// TIA Portal project "PLC" (V15.1)

(* hardware
DEVICE "S7-1200 station_1"  S7-1200 Station
   slot 0: "Rack_0"  S7-1200 Rack  Rack  V1.0
   slot 1: "PLC_1"  CPU 1214C DC/DC/DC  6ES7 214-1AG40-0XB0  V4.2
DEVICE "HMI_1"  KTP700 Basic PN
   slot 0: "HMI_1"  KTP700 Basic PN  6AV2 123-2GB03-0AX0  15.1.0.0
   slot 1: "HMI_RT_1"  KTP700 Basic PN  6AV2 123-2GB03-0AX0  15.1.0.0
   slot 5: "HMI_1.IE_CP_1"  PROFINET Interface  15.0.1.0
      slot 1: "PROFINET Interface_1"  PROFINET Interface
         slot 1: "Port_1"  Port
*)

// ===== PLC "PLC_1"  CPU 1214C DC/DC/DC =====

VAR_GLOBAL   // PLC tag table "默认变量表"
   "物料到位信号" AT %I0.0 : Bool;
   "物料检测信号" AT %I0.6 : Bool;
   "传送带正转信号" AT %Q0.1 : Bool;
   "推料动作" AT %Q0.4 : Bool;
   "运行步骤" AT %MW100 : Int;
   "物资发放" AT %M22.7 : Bool;
END_VAR

DATA_BLOCK "人脸语音通讯"   // DB9
{ S7_Optimized_Access := 'TRUE' }
VERSION : 0.1
   VAR
      re_data : Array[0..31] of Byte;
      use_data : Array[0..31] of String;
      empty_data : Array[0..31] of Byte;
      人脸语音通讯成功 : Bool;
   END_VAR
BEGIN
END_DATA_BLOCK

DATA_BLOCK "图像识别通讯"   // DB12
{ S7_Optimized_Access := 'TRUE' }
VERSION : 0.1
   VAR
      re_data : Array[0..31] of Byte;
      use_data : Array[0..31] of String;
      empty_data : Array[0..31] of Byte;
      tx_data : Array[0..31] of Byte;
      人员1信息 : Array[0..6] of String;
      人员2信息 : Array[0..6] of String;
      人员3信息 : Array[0..6] of String;
      人员4信息 : Array[0..6] of String;
      人员5信息 : Array[0..6] of String;
      人员6信息 : Array[0..6] of String;
      图像识别发送标志位 : Bool;
      图像识别通讯成功 : Bool;
   END_VAR
BEGIN
END_DATA_BLOCK

DATA_BLOCK "视觉通讯"   // DB15
{ S7_Optimized_Access := 'TRUE' }
VERSION : 0.1
   VAR
      re_data : Array[0..310] of Byte;
      use_data : Array[0..100] of String;
      empty_data : Array[0..310] of Byte;
      tx_data : Array[0..310] of Byte;
      发送数据的长度 : Int;
      视觉发送标志位 : Bool;
      视觉通讯成功 : Bool;
      A地区状态 : String;
      B地区状态 : String;
      C地区状态 : String;
      D地区状态 : String;
   END_VAR
BEGIN
END_DATA_BLOCK

DATA_BLOCK "机器人通讯"   // DB18
{ S7_Optimized_Access := 'TRUE' }
VERSION : 0.1
   VAR
      re_data : Array[0..31] of Byte;
      use_data : Array[0..31] of String;
      empty_data : Array[0..31] of Byte;
      tx_data : Array[0..31] of Byte;
      机器人发送标志位 : Bool;
      机器人通讯成功 : Bool;
      二维码分类计数 : Int;
   END_VAR
BEGIN
END_DATA_BLOCK

// folder: System blocks/Program resources

DATA_BLOCK "PLC_1_Receive_DB"   // DB1
{ S7_Optimized_Access := 'TRUE' }
AUTHOR : SIMATIC
FAMILY : MC7Plus
NAME : TC_IP_v4
VERSION : 1.0
// stored: InstanceOfName TCON_IP_v4
"TCON_IP_v4"
BEGIN
   ID := 1;
   InterfaceId := 64;
   LocalPort := 4001;
END_DATA_BLOCK

DATA_BLOCK "PLC_1_Receive_DB_1"   // DB2
{ S7_Optimized_Access := 'TRUE' }
AUTHOR : SIMATIC
FAMILY : MC7Plus
NAME : TC_IP_v4
VERSION : 1.0
// stored: InstanceOfName TCON_IP_v4
"TCON_IP_v4"
BEGIN
   ID := 2;
   InterfaceId := 64;
   LocalPort := 2005;
END_DATA_BLOCK

DATA_BLOCK "PLC_1_Receive_DB_2"   // DB3
{ S7_Optimized_Access := 'TRUE' }
AUTHOR : SIMATIC
FAMILY : MC7Plus
NAME : TC_IP_v4
VERSION : 1.0
// stored: InstanceOfName TCON_IP_v4
"TCON_IP_v4"
BEGIN
   ID := 3;
   InterfaceId := 64;
   LocalPort := 3001;
END_DATA_BLOCK

DATA_BLOCK "PLC_1_Receive_DB_3"   // DB4
{ S7_Optimized_Access := 'TRUE' }
AUTHOR : SIMATIC
FAMILY : MC7Plus
NAME : TC_IP_v4
VERSION : 1.0
// stored: InstanceOfName TCON_IP_v4
"TCON_IP_v4"
BEGIN
   ID := 4;
   InterfaceId := 64;
   LocalPort := 2001;
END_DATA_BLOCK

DATA_BLOCK "延时函数"   // DB13
{ S7_Optimized_Access := 'TRUE' }
AUTHOR : Simatic
FAMILY : IEC
NAME : IEC_TMR
VERSION : 1.0
// stored: InstanceOfName IEC_TIMER
"IEC_TIMER"
BEGIN
END_DATA_BLOCK

// folder: (top level)

FUNCTION "发送" : Void   // FC2, SCL
{ S7_Optimized_Access := 'TRUE' }
VERSION : 0.1
   VAR_INPUT
      buf : String;
      num : Int;
   END_VAR
   VAR_TEMP
      strlen : Int;
   END_VAR
BEGIN
   //字符串转换成字符指令
   "视觉通讯".发送数据的长度 := LEN(#buf);
   IF #num = 2 THEN
       Strg_TO_Chars(Strg := #buf,  //需要转换的字符串
                     pChars := 0,    //字符数组的起始位置
                     Cnt => #strlen, // 转成成功的长度，储存到
                     Chars := "图像识别通讯".tx_data);//字符串的数组
       "图像识别通讯".图像识别发送标志位 := 1;
   ELSIF #num = 3 THEN
       Strg_TO_Chars(Strg := #buf,
                     pChars := 0,
                     Cnt => #strlen,
                     Chars := "视觉通讯".tx_data);
       "视觉通讯".视觉发送标志位 := 1;
   ELSIF #num = 4 THEN
       Strg_TO_Chars(Strg := #buf,
                     pChars := 0,
                     Cnt => #strlen,
                     Chars := "机器人通讯".tx_data);
       "机器人通讯".机器人发送标志位 := 1;
   END_IF;
END_FUNCTION

FUNCTION "图像识别通讯主程序" : Void   // FC4, LAD
{ S7_Optimized_Access := 'TRUE' }
VERSION : 0.1
   VAR_TEMP
      i : Int;
      i_1 : Int;
      i_2 : Int;
      send_data : String;
   END_VAR
BEGIN

REGION Network 1
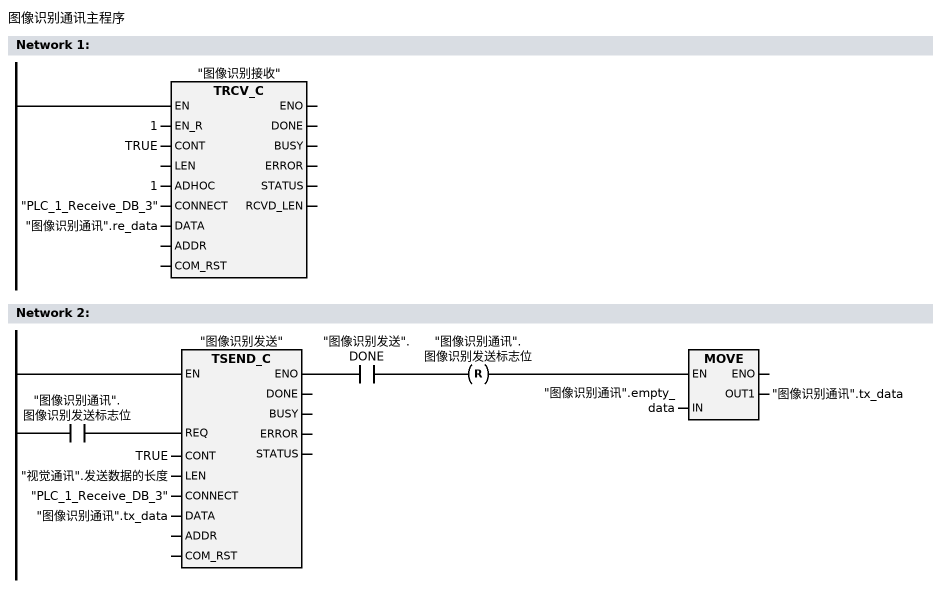
   "图像识别接收"(EN_R := 1, CONT := TRUE, ADHOC := 1, CONNECT := "PLC_1_Receive_DB_3", DATA := "图像识别通讯".re_data);   // TRCV_C
END_REGION

REGION Network 2
   // ENO of a box is taken as its EN; it also drops when the box reports an error
   "图像识别发送"(REQ := "图像识别通讯".图像识别发送标志位,   // TSEND_C
            CONT := TRUE,
            LEN := "视觉通讯".发送数据的长度,
            CONNECT := "PLC_1_Receive_DB_3",
            DATA := "图像识别通讯".tx_data);
   IF "图像识别发送".DONE THEN
       "图像识别通讯".图像识别发送标志位 := FALSE;
       "图像识别通讯".tx_data := "图像识别通讯".empty_data;
   END_IF;
END_REGION

REGION Network 3 (SCL)
   IF "图像识别接收".DONE THEN
       //字符分割函数
       FOR #i := 0 TO 31 DO
           IF "图像识别通讯".re_data[#i] = ',' OR "图像识别通讯".re_data[#i] = 16#0 THEN
               Chars_TO_Strg(Chars := "图像识别通讯".re_data,
                             pChars := #i_1,
                             Cnt := #i - #i_1,
                             Strg => "图像识别通讯".use_data[#i_2]);
               #i_1 := #i + 1;
               #i_2 += 1;
           END_IF;
       END_FOR;
       "图像识别通讯".re_data := "图像识别通讯".empty_data;

       FOR #i := 0 TO 2 DO
           IF "图像识别通讯".use_data[0] = "图像识别通讯"."人员1信息"[#i + 2] THEN
               "发送"(buf := 'D1',
                    num := 4);
               EXIT;
           END_IF;
           IF "图像识别通讯".use_data[0] = "图像识别通讯"."人员2信息"[#i + 2] THEN
               //"视觉通讯"."2号人员信息"[#i + 2] := ' ';
               "发送"(buf := 'A1',
                     num := 4);
               EXIT;
           END_IF;
           IF "图像识别通讯".use_data[0] = "图像识别通讯"."人员3信息"[#i + 2] THEN
               //"视觉通讯"."3号人员信息"[#i + 2] := ' ';
               "发送"(buf := 'B1',
                    num := 4);
               EXIT;
           END_IF;
           IF "图像识别通讯".use_data[0] = "图像识别通讯"."人员4信息"[#i + 2] THEN
               //"视觉通讯"."4号人员信息"[#i + 2] := ' ';
               "发送"(buf := 'C1',
                    num := 4);
               EXIT;
           END_IF;
       END_FOR;
   END_IF;
END_REGION
END_FUNCTION

FUNCTION "机器人通讯主程序" : Void   // FC5, LAD
{ S7_Optimized_Access := 'TRUE' }
VERSION : 0.1
   VAR_TEMP
      i : Int;
      i_1 : Int;
      i_2 : Int;
      ab : String;
   END_VAR
BEGIN

REGION Network 1
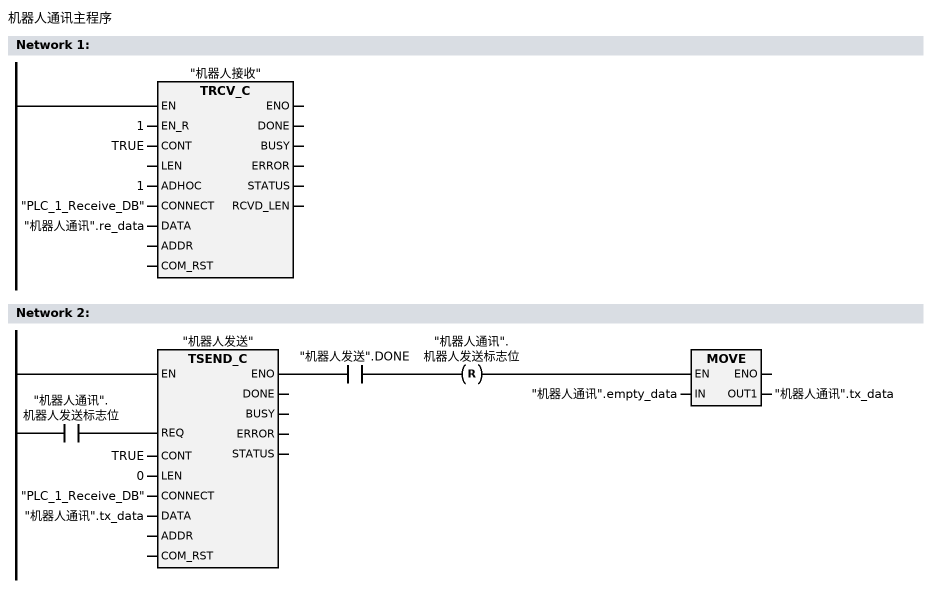
   "机器人接收"(EN_R := 1, CONT := TRUE, ADHOC := 1, CONNECT := "PLC_1_Receive_DB", DATA := "机器人通讯".re_data);   // TRCV_C
END_REGION

REGION Network 2
   // ENO of a box is taken as its EN; it also drops when the box reports an error
   "机器人发送"(REQ := "机器人通讯".机器人发送标志位,   // TSEND_C
           CONT := TRUE,
           LEN := 0,
           CONNECT := "PLC_1_Receive_DB",
           DATA := "机器人通讯".tx_data);
   IF "机器人发送".DONE THEN
       "机器人通讯".机器人发送标志位 := FALSE;
       "机器人通讯".tx_data := "机器人通讯".empty_data;
   END_IF;
END_REGION

REGION Network 3 (SCL)
   IF "机器人接收".DONE THEN
       //字符分割函数
       FOR #i := 0 TO 31 DO
           IF "机器人通讯".re_data[#i] = ',' OR "机器人通讯".re_data[#i] = 16#0 THEN
               Chars_TO_Strg(Chars := "机器人通讯".re_data,
                             pChars := #i_1,
                             Cnt := #i - #i_1,
                             Strg => "机器人通讯".use_data[#i_2]);
               #i_1 := #i + 1;
               #i_2 += 1;
           END_IF;
       END_FOR;
       "机器人通讯".re_data := "机器人通讯".empty_data;
       //二维码分类
       IF "机器人通讯".use_data[0] = 'ok1' THEN
           "发送"(buf := 'ewm',
                num := 3);
       ELSIF "机器人通讯".use_data[0] = 'ok2' THEN
           IF "机器人通讯".二维码分类计数 > 4 THEN
               ;
           ELSE
               "机器人通讯".二维码分类计数 += 1;
               "发送"(buf := 'set',
                    num := 4);
           END_IF;
       ELSIF "机器人通讯".use_data[0] = 'run' THEN
           "物资发放" := 1;
       END_IF;
   END_IF;
END_REGION
END_FUNCTION

FUNCTION "视觉通讯主程序" : Void   // FC6, LAD
{ S7_Optimized_Access := 'TRUE' }
VERSION : 0.1
   VAR_TEMP
      i : Int;
      i_1 : Int;
      i_2 : Int;
   END_VAR
BEGIN

REGION Network 1
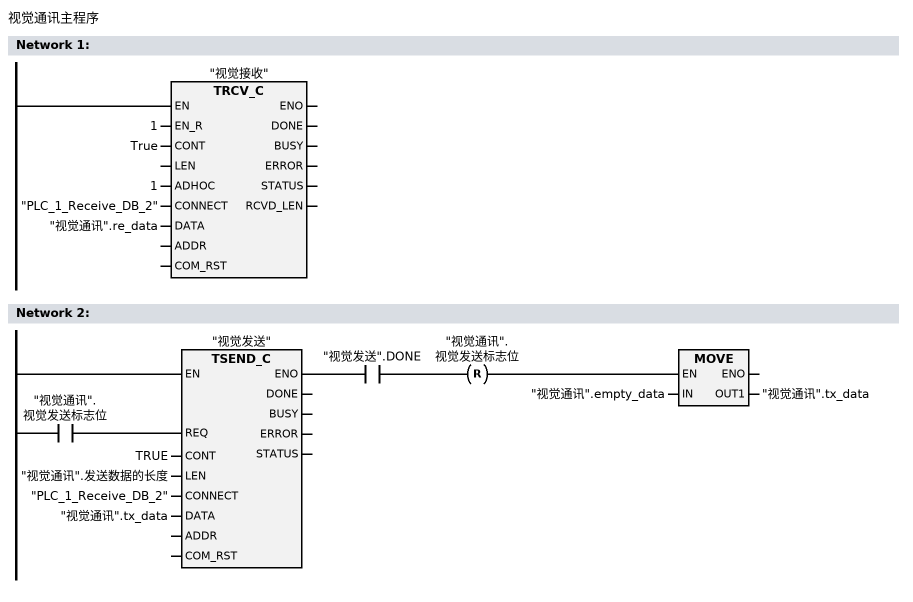
   "视觉接收"(EN_R := 1, CONT := True, ADHOC := 1, CONNECT := "PLC_1_Receive_DB_2", DATA := "视觉通讯".re_data);   // TRCV_C
END_REGION

REGION Network 2
   // ENO of a box is taken as its EN; it also drops when the box reports an error
   "视觉发送"(REQ := "视觉通讯".视觉发送标志位,   // TSEND_C
          CONT := TRUE,
          LEN := "视觉通讯".发送数据的长度,
          CONNECT := "PLC_1_Receive_DB_2",
          DATA := "视觉通讯".tx_data);
   IF "视觉发送".DONE THEN
       "视觉通讯".视觉发送标志位 := FALSE;
       "视觉通讯".tx_data := "视觉通讯".empty_data;
   END_IF;
END_REGION

REGION Network 3 (SCL)
   IF "视觉接收".DONE THEN
       //字符分割函数
       FOR #i := 0 TO 310 DO
           IF "视觉通讯".re_data[#i] = ',' OR "视觉通讯".re_data[#i] = 16#0 THEN
               Chars_TO_Strg(Chars := "视觉通讯".re_data,
                             pChars := #i_1,
                             Cnt := #i - #i_1,
                             Strg => "视觉通讯".use_data[#i_2]);
               #i_1 := #i + 1;
               #i_2 += 1;
           END_IF;
       END_FOR;
       "视觉通讯".re_data := "视觉通讯".empty_data;

       //处理地图信息

       IF "视觉通讯".use_data[0] = '{name:Tom;active:A;drink:kuangquanshui;food:fangbianmian;supplies:xifashui}' THEN
           "图像识别通讯".人员1信息[0] := 'Tom';
           "图像识别通讯".人员1信息[1] := 'A';
           "图像识别通讯".人员1信息[2] := 'kuangquanshui';
           "图像识别通讯".人员1信息[3] := 'fangbianmian';
           "图像识别通讯".人员1信息[4] := 'xifashui';
           "发送"(buf := 'D1',
                num := 4);
       ELSIF "视觉通讯".use_data[0] = '{name:Jack;active:B;drink:kele;food:pingguo;supplies:maojin}' THEN
           "图像识别通讯".人员2信息[0] := 'Jack';
           "图像识别通讯".人员2信息[1] := 'B';
           "图像识别通讯".人员2信息[2] := 'kele';
           "图像识别通讯".人员2信息[3] := 'pingguo';
           "图像识别通讯".人员2信息[4] := 'maojin';
           "发送"(buf:='A1',
                num:= 4);

           //处理物资的坐标信息

       ELSIF "视觉通讯".use_data[0] = '{name:Andy;active:C;drink:fenda;food:mianbao;supplies:yagao}' THEN
           "图像识别通讯".人员3信息[0] := 'Andy';
           "图像识别通讯".人员3信息[1] := 'C';
           "图像识别通讯".人员3信息[2] := 'fenda';
           "图像识别通讯".人员3信息[3] := 'mianbao';
           "图像识别通讯".人员3信息[4] := 'yagao';
           "发送"(buf := 'B1',
                num := 4);
       ELSIF "视觉通讯".use_data[0] = '{name:Vicky;active:D;drink:xuebi;food:guantou;supplies:zhijin}' THEN
           "图像识别通讯".人员4信息[0] := 'Vicky';
           "图像识别通讯".人员4信息[1] := 'D';
           "图像识别通讯".人员4信息[2] := 'xuebi';
           "图像识别通讯".人员4信息[3] := 'guantou';
           "图像识别通讯".人员4信息[4] := 'zhijin';
           "发送"(buf := 'C1',
                num := 4);
       ELSIF "视觉通讯".use_data[0] = '{name:Cindy;active:E;drink:hongniu;food:mangguo;supplies:tuoxie}' THEN
           "图像识别通讯".人员5信息[0] := 'Cindy';
           "图像识别通讯".人员5信息[1] := 'E';
           "图像识别通讯".人员5信息[2] := 'hongniu';
           "图像识别通讯".人员5信息[3] := 'mangguo';
           "图像识别通讯".人员5信息[4] := 'tuoxie';
           "发送"(buf := 'return',
                num := 4);
       ELSIF "视觉通讯".use_data[0] = '{name:David;active:F;drink:kuangquanshui;food:xiangchang;supplies:xiangzao}' THEN
           "图像识别通讯".人员6信息[0] := 'David';
           "图像识别通讯".人员6信息[1] := 'F';
           "图像识别通讯".人员6信息[2] := 'kuangquanshui';
           "图像识别通讯".人员6信息[3] := 'xiangchang';
           "图像识别通讯".人员6信息[4] := 'xiangzao';
           "发送"(buf := 'return',
                num := 4);
       ELSIF "视觉通讯".use_data[0] = 'geli' THEN
           "视觉通讯".A地区状态 := 'geli';
           "视觉通讯".B地区状态 := 'low';
           "视觉通讯".C地区状态 := 'mid';
           "视觉通讯".D地区状态 := 'high';

       ELSIF "视觉通讯".use_data[0] = 'image' THEN
           "发送"(buf := 'verify',
                num := 2);
       ELSIF "视觉通讯".use_data[0] = 'kong' THEN
           "发送"(buf := 'F2',
                num := 4);

       END_IF;
   END_IF;
END_REGION
END_FUNCTION

FUNCTION "人脸语音通讯主程序" : Void   // FC7, LAD
{ S7_Optimized_Access := 'TRUE' }
VERSION : 0.1
   VAR_TEMP
      i : Int;
      i_1 : Int;
      i_2 : Int;
   END_VAR
   VAR_TEMP   // added for the SCL form of the ladder/FBD networks
      _w1 : Bool;
      _w2 : Bool;
   END_VAR
BEGIN

REGION Network 1
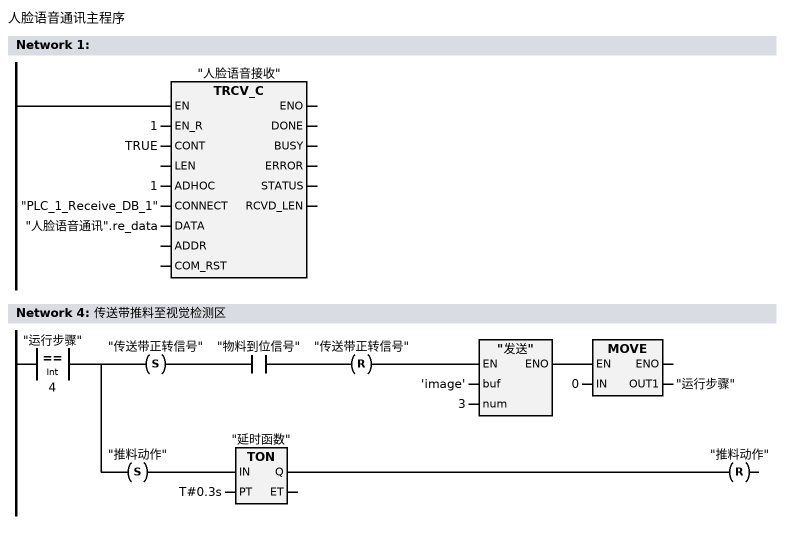
   "人脸语音接收"(EN_R := 1, CONT := TRUE, ADHOC := 1, CONNECT := "PLC_1_Receive_DB_1", DATA := "人脸语音通讯".re_data);   // TRCV_C
END_REGION

REGION Network 2 (SCL)
   IF "人脸语音接收".DONE THEN
       //字符分割函数
       FOR #i := 0 TO 31 DO
           IF "人脸语音通讯".re_data[#i] = ',' OR "人脸语音通讯".re_data[#i] = 16#00 THEN
               Chars_TO_Strg(Chars := "人脸语音通讯".re_data,
                             pChars := #i_1,
                             Cnt := #i - #i_1,
                             Strg => "人脸语音通讯".use_data[#i_2]);
               #i_1 := #i + 1;
               #i_2 += 1;
           END_IF;
       END_FOR;
       "人脸语音通讯".re_data := "人脸语音通讯".empty_data;

       IF "人脸语音通讯".use_data[0] = 'guankong' THEN
           "发送"(buf := 'set',
                num := 4);
       ELSIF "人脸语音通讯".use_data[0] = 'fafang' THEN
           "物资发放" := 1;
       ELSIF "人脸语音通讯".use_data[0] = 'A' THEN
           "发送"(buf := 'A',
                num := 3);
       END_IF;
   END_IF;
END_REGION

REGION Network 3 (SCL)
   IF "物资发放" AND "物料检测信号" THEN
       "运行步骤" := 4;
       "物资发放" := 0;
   END_IF;
END_REGION

REGION Network 4: 传送带推料至视觉检测区
   #_w1 := "运行步骤" = 4;
   IF #_w1 THEN "传送带正转信号" := TRUE; END_IF;
   IF #_w1 AND "物料到位信号" THEN "传送带正转信号" := FALSE; END_IF;
   "发送"(EN := #_w1 AND "物料到位信号", buf := 'image', num := 3, ENO => #_w2);
   IF #_w2 THEN "运行步骤" := 0; END_IF;
   IF #_w1 THEN "推料动作" := TRUE; END_IF;
   "延时函数".TON(IN := #_w1, PT := T#0.3s);
   IF "延时函数".Q THEN "推料动作" := FALSE; END_IF;
END_REGION
END_FUNCTION

ORGANIZATION_BLOCK "Main"   // OB1, LAD, ProgramCycle
TITLE = "Main Program Sweep (Cycle)"
{ S7_Optimized_Access := 'TRUE' }
VERSION : 0.1
   VAR_INPUT
      Initial_Call : Bool;   // Initial call of this OB
      Remanence : Bool;   // =True, if remanent data are available
   END_VAR
   VAR_TEMP
      i : Int;
      data : String;
   END_VAR
BEGIN

REGION Network 1: 推料
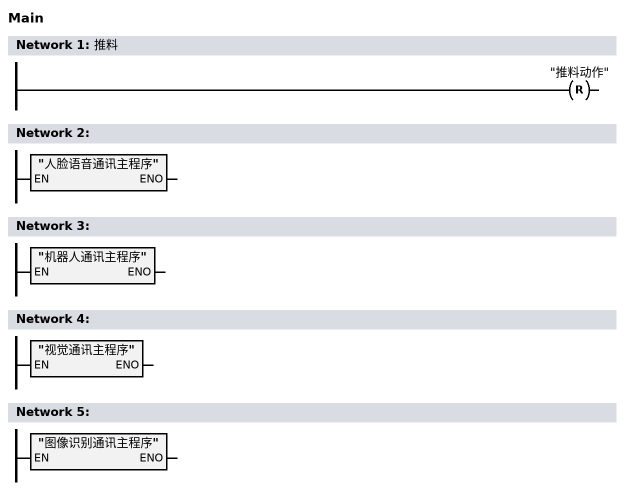
   RUNG wire#powerrail
      R_Coil( "推料动作" )
   END_RUNG
   // the same network as SCL:
   "推料动作" := FALSE;
END_REGION

REGION Network 2
   RUNG wire#powerrail
      "人脸语音通讯主程序"()
   END_RUNG
   // the same network as SCL:
   "人脸语音通讯主程序"();
END_REGION

REGION Network 3
   RUNG wire#powerrail
      "机器人通讯主程序"()
   END_RUNG
   // the same network as SCL:
   "机器人通讯主程序"();
END_REGION

REGION Network 4
   RUNG wire#powerrail
      "视觉通讯主程序"()
   END_RUNG
   // the same network as SCL:
   "视觉通讯主程序"();
END_REGION

REGION Network 5
   RUNG wire#powerrail
      "图像识别通讯主程序"()
   END_RUNG
   // the same network as SCL:
   "图像识别通讯主程序"();
END_REGION
END_ORGANIZATION_BLOCK

(* ===== HMI "HMI_RT_1" =====
system functions are stored by id; their names below are inferred from use
connection "HMI_连接_1": ETHERNET, SMART_S7_1200_OMS

HMI tags "默认变量表"
   "视觉通讯_A地区状态" : String[254] = PLC 视觉通讯.A地区状态, 1 s
   "视觉通讯_B地区状态" : String[254] = PLC 视觉通讯.B地区状态, 1 s
   "视觉通讯_C地区状态" : String[254] = PLC 视觉通讯.C地区状态, 1 s
   "视觉通讯_D地区状态" : String[254] = PLC 视觉通讯.D地区状态, 1 s
   "图像识别通讯_人员1信息{0}" : String[254] = PLC 图像识别通讯.人员1信息[0], 1 s
   "图像识别通讯_人员1信息{1}" : String[254] = PLC 图像识别通讯.人员1信息[1], 1 s
   "图像识别通讯_人员1信息{2}" : String[254] = PLC 图像识别通讯.人员1信息[2], 1 s
   "图像识别通讯_人员1信息{4}" : String[254] = PLC 图像识别通讯.人员1信息[4], 1 s
   "图像识别通讯_人员1信息{3}" : String[254] = PLC 图像识别通讯.人员1信息[3], 1 s
   "图像识别通讯_人员2信息{0}" : String[254] = PLC 图像识别通讯.人员2信息[0], 1 s
   "图像识别通讯_人员2信息{1}" : String[254] = PLC 图像识别通讯.人员2信息[1], 1 s
   "图像识别通讯_人员2信息{2}" : String[254] = PLC 图像识别通讯.人员2信息[2], 1 s
   "图像识别通讯_人员2信息{3}" : String[254] = PLC 图像识别通讯.人员2信息[3], 1 s
   "图像识别通讯_人员2信息{4}" : String[254] = PLC 图像识别通讯.人员2信息[4], 1 s
   "图像识别通讯_人员3信息{0}" : String[254] = PLC 图像识别通讯.人员3信息[0], 1 s
   "图像识别通讯_人员3信息{1}" : String[254] = PLC 图像识别通讯.人员3信息[1], 1 s
   "图像识别通讯_人员3信息{2}" : String[254] = PLC 图像识别通讯.人员3信息[2], 1 s
   "图像识别通讯_人员3信息{3}" : String[254] = PLC 图像识别通讯.人员3信息[3], 1 s
   "图像识别通讯_人员3信息{4}" : String[254] = PLC 图像识别通讯.人员3信息[4], 1 s
   "图像识别通讯_人员4信息{0}" : String[254] = PLC 图像识别通讯.人员4信息[0], 1 s
   "图像识别通讯_人员4信息{1}" : String[254] = PLC 图像识别通讯.人员4信息[1], 1 s
   "图像识别通讯_人员4信息{2}" : String[254] = PLC 图像识别通讯.人员4信息[2], 1 s
   "图像识别通讯_人员4信息{3}" : String[254] = PLC 图像识别通讯.人员4信息[3], 1 s
   "图像识别通讯_人员4信息{4}" : String[254] = PLC 图像识别通讯.人员4信息[4], 1 s
   "图像识别通讯_人员5信息{0}" : String[254] = PLC 图像识别通讯.人员5信息[0], 1 s
   "图像识别通讯_人员5信息{1}" : String[254] = PLC 图像识别通讯.人员5信息[1], 1 s
   "图像识别通讯_人员5信息{2}" : String[254] = PLC 图像识别通讯.人员5信息[2], 1 s
   "图像识别通讯_人员5信息{3}" : String[254] = PLC 图像识别通讯.人员5信息[3], 1 s
   "图像识别通讯_人员5信息{4}" : String[254] = PLC 图像识别通讯.人员5信息[4], 1 s
   "图像识别通讯_人员6信息{0}" : String[254] = PLC 图像识别通讯.人员6信息[0], 1 s
   "图像识别通讯_人员6信息{1}" : String[254] = PLC 图像识别通讯.人员6信息[1], 1 s
   "图像识别通讯_人员6信息{2}" : String[254] = PLC 图像识别通讯.人员6信息[2], 1 s
   "图像识别通讯_人员6信息{3}" : String[254] = PLC 图像识别通讯.人员6信息[3], 1 s
   "图像识别通讯_人员6信息{4}" : String[254] = PLC 图像识别通讯.人员6信息[4], 1 s

Template "模板_1" 800x480
   Button "退出" at 714,429 size 71x50; TextOff '退出'; PictureOff "ExitRuntime_KTP700_Basic_PN_TR"; PictureOn "ExitRuntime_KTP700_Basic_PN_TR"
      on Release: StopRuntime(0)
   Button "Template_Button" at 614,429 size 71x50; TextOff 'Text'
   Button "Template_Button_1" at 514,429 size 71x50; TextOff 'Text'
   Button "Template_Button_2" at 414,429 size 71x50; TextOff 'Text'
   Button "Template_Button_3" at 314,429 size 71x50; TextOff 'Text'
   Button "Template_Button_4" at 214,429 size 71x50; TextOff 'Text'
   Button "Template_Button_5" at 114,429 size 71x50; TextOff 'Text'
   Button "起始画面" at 14,429 size 71x50; TextOff '起始画面'; PictureOff "NavigateHome_KTP700_Basic_PN_TR"; PictureOn "NavigateHome_KTP700_Basic_PN_TR"
      on Release: ActivateScreen("主界面", 0)
   DateTimeField "HmiScreenItemData" at 695,25 size 105x25
   DateTimeField "HmiScreenItemData_1" at 695,0 size 105x25
   GraphicView "Logo" at 0,0 size 91x51; Picture "HMI_1 的 Logo"

screen "主界面" 800x480
   TextField "文本域_1" at 283,10 size 221x39; Text '信息监控界面'
   TextField "文本域_2" at 45,140 size 173x27; Text '各小区疫情信息'
   TextField "文本域_3" at 461,75 size 149x27; Text '人员信息采集'
   TextField "文本域_4" at 40,204 size 82x20; Text '第一小区:'
   TextField "文本域_5" at 40,253 size 82x20; Text '第二小区:'
   TextField "文本域_6" at 40,301 size 82x20; Text '第三小区:'
   TextField "文本域_7" at 40,348 size 82x20; Text '第四小区:'
   TextField "文本域_8" at 304,119 size 39x20; Text '姓名'
   IOField "I/O 域_1" at 296,150 size 55x32; FormatPattern ????????????????????????????????????????????????????????????????????????????????
      ProcessValue <- "图像识别通讯_人员1信息{0}"
   IOField "I/O 域_2" at 296,202 size 56x32; FormatPattern ????????????????????????????????????????????????????????????????????????????????
      ProcessValue <- "图像识别通讯_人员2信息{0}"
   IOField "I/O 域_3" at 295,254 size 58x32; FormatPattern ????????????????????????????????????????????????????????????????????????????????
      ProcessValue <- "图像识别通讯_人员3信息{0}"
   IOField "I/O 域_4" at 295,306 size 58x32; FormatPattern ????????????????????????????????????????????????????????????????????????????????
      ProcessValue <- "图像识别通讯_人员4信息{0}"
   TextField "文本域_9" at 396,119 size 39x20; Text '行程'
   IOField "I/O 域_5" at 401,150 size 31x32; FormatPattern ????????????????????????????????????????????????????????????????????????????????
      ProcessValue <- "图像识别通讯_人员1信息{1}"
   TextField "文本域_10" at 492,119 size 39x20; Text '饮品'
   IOField "I/O 域_9" at 469,150 size 84x32; FormatPattern ????????????????????????????????????????????????????????????????????????????????
      ProcessValue <- "图像识别通讯_人员1信息{2}"
   IOField "I/O 域_6" at 401,202 size 31x32; FormatPattern ????????????????????????????????????????????????????????????????????????????????
      ProcessValue <- "图像识别通讯_人员2信息{1}"
   IOField "I/O 域_7" at 401,254 size 31x32; FormatPattern ????????????????????????????????????????????????????????????????????????????????
      ProcessValue <- "图像识别通讯_人员3信息{1}"
   IOField "I/O 域_8" at 401,306 size 31x32; FormatPattern ????????????????????????????????????????????????????????????????????????????????
      ProcessValue <- "图像识别通讯_人员4信息{1}"
   IOField "I/O 域_10" at 469,202 size 84x32; FormatPattern ????????????????????????????????????????????????????????????????????????????????
      ProcessValue <- "图像识别通讯_人员2信息{2}"
   IOField "I/O 域_11" at 469,254 size 84x32; FormatPattern ????????????????????????????????????????????????????????????????????????????????
      ProcessValue <- "图像识别通讯_人员3信息{2}"
   IOField "I/O 域_12" at 469,306 size 84x32; FormatPattern ????????????????????????????????????????????????????????????????????????????????
      ProcessValue <- "图像识别通讯_人员4信息{2}"
   TextField "文本域_11" at 597,119 size 39x20; Text '食物'
   IOField "I/O 域_13" at 574,150 size 84x32; FormatPattern ????????????????????????????????????????????????????????????????????????????????
      ProcessValue <- "图像识别通讯_人员1信息{3}"
   IOField "I/O 域_14" at 574,202 size 84x32; FormatPattern ????????????????????????????????????????????????????????????????????????????????
      ProcessValue <- "图像识别通讯_人员2信息{3}"
   IOField "I/O 域_15" at 574,254 size 84x32; FormatPattern ????????????????????????????????????????????????????????????????????????????????
      ProcessValue <- "图像识别通讯_人员3信息{3}"
   IOField "I/O 域_16" at 574,306 size 84x32; FormatPattern ????????????????????????????????????????????????????????????????????????????????
      ProcessValue <- "图像识别通讯_人员4信息{3}"
   TextField "文本域_12" at 683,119 size 73x20; Text '日常用品'
   IOField "I/O 域_17" at 677,150 size 84x32; FormatPattern ????????????????????????????????????????????????????????????????????????????????
      ProcessValue <- "图像识别通讯_人员1信息{4}"
   IOField "I/O 域_18" at 677,202 size 84x32; FormatPattern ????????????????????????????????????????????????????????????????????????????????
      ProcessValue <- "图像识别通讯_人员2信息{4}"
   IOField "I/O 域_19" at 677,254 size 84x32; FormatPattern ????????????????????????????????????????????????????????????????????????????????
      ProcessValue <- "图像识别通讯_人员3信息{4}"
   IOField "I/O 域_20" at 677,306 size 84x32; FormatPattern ????????????????????????????????????????????????????????????????????????????????
      ProcessValue <- "图像识别通讯_人员4信息{4}"
   IOField "I/O 域_21" at 134,199 size 55x32; FormatPattern ????????????????????????????????????????????????????????????????????????????????
      ProcessValue <- "视觉通讯_A地区状态"
   IOField "I/O 域_22" at 134,248 size 55x32; FormatPattern ????????????????????????????????????????????????????????????????????????????????
      ProcessValue <- "视觉通讯_B地区状态"
   IOField "I/O 域_23" at 134,296 size 55x32; FormatPattern ????????????????????????????????????????????????????????????????????????????????
      ProcessValue <- "视觉通讯_C地区状态"
   IOField "I/O 域_24" at 134,343 size 55x32; FormatPattern ????????????????????????????????????????????????????????????????????????????????
      ProcessValue <- "视觉通讯_D地区状态"
   IOField "I/O 域_25" at 295,358 size 58x32; FormatPattern ????????????????????????????????????????????????????????????????????????????????
      ProcessValue <- "图像识别通讯_人员5信息{0}"
   IOField "I/O 域_26" at 401,358 size 31x32; FormatPattern ????????????????????????????????????????????????????????????????????????????????
      ProcessValue <- "图像识别通讯_人员5信息{1}"
   IOField "I/O 域_27" at 469,358 size 84x32; FormatPattern ????????????????????????????????????????????????????????????????????????????????
      ProcessValue <- "图像识别通讯_人员5信息{2}"
   IOField "I/O 域_28" at 574,358 size 84x32; FormatPattern ????????????????????????????????????????????????????????????????????????????????
      ProcessValue <- "图像识别通讯_人员5信息{3}"
   IOField "I/O 域_29" at 677,358 size 84x32; FormatPattern ????????????????????????????????????????????????????????????????????????????????
      ProcessValue <- "图像识别通讯_人员5信息{4}"
   IOField "I/O 域_30" at 295,410 size 58x32; FormatPattern ????????????????????????????????????????????????????????????????????????????????
      ProcessValue <- "图像识别通讯_人员6信息{0}"
   IOField "I/O 域_31" at 401,410 size 31x32; FormatPattern ????????????????????????????????????????????????????????????????????????????????
      ProcessValue <- "图像识别通讯_人员6信息{1}"
   IOField "I/O 域_32" at 469,410 size 84x32; FormatPattern ????????????????????????????????????????????????????????????????????????????????
      ProcessValue <- "图像识别通讯_人员6信息{2}"
   IOField "I/O 域_33" at 574,410 size 84x32; FormatPattern ????????????????????????????????????????????????????????????????????????????????
      ProcessValue <- "图像识别通讯_人员6信息{3}"
   IOField "I/O 域_34" at 677,410 size 84x32; FormatPattern ????????????????????????????????????????????????????????????????????????????????
      ProcessValue <- "图像识别通讯_人员6信息{4}"
*)